FUNCTION_BLOCK FB_Zuiger
VAR_INPUT
	i_eState 			: eSingleState;
	i_eModes			: eModus;
	i_xMoveCiliderDown	: BOOL;
	i_xHallSensorIn		: BOOL;
	i_xHallSensorOut	: BOOL;
	i_xEndSwitchIn		: BOOL;
	i_xEndSwitchOut		: BOOL;
	i_rPressureSensor	: REAL; 
	i_xAlarmResetCilinder	: BOOL;
	i_xAlarmResetAlarmHorizontalMovement	: BOOL;
	i_xAlarmResetPressure : BOOL;
	i_xButtonManStopall : BOOL;
	eManCiliderPosition		: eZuigerCilinderposition;
	eManHorizotalPosition	: eZuigerHorizontaal;
	i_xButtonManVacumOn	: BOOL;
END_VAR
VAR_OUTPUT
	o_xMotor 					: BOOL := FALSE;
	o_xMotorDirectionOut		: BOOL;
	o_xErrorHorizontalMovement 	: BOOL := FALSE;
	o_xAlarmHorizontalMovement	: BOOL;
	o_xMagnetValveCilinder		: BOOL := FALSE;
	o_xMagnetValveVacum	: 			BOOL := FALSE;
	o_xErrorCilinder			: BOOL := FALSE;
	o_xAlarmCilinder			: BOOL;
	o_xErrorPressure			: BOOL := FALSE;
	o_xAlarmPressure			: BOOL;
	o_eCiliderPosition			: eZuigerCilinderposition;
	o_eHorizotalPosition		: eZuigerHorizontaal;
END_VAR
VAR
	eWistedCiliderPosition		: eZuigerCilinderposition;
	eWistedHorizotalPosition	: eZuigerHorizontaal;
	istepcycel : INT;
	TimerCilinder : TON;
	timTimerValue : TIME := T#10S;
	xTimerCilinderRunning: BOOL;
	TimerHorizontal : TON;
	xTimerHorizontalRunning: BOOL;
	
	rPressure_bar: REAL ;
	rMaxbarsensor: REAL := 6;
	rlowpressure: REAL := 4;
	
	
	SIMFUNCTIONING : BOOL := 1;
	o_sStateString: STRING(30);
END_VAR

//Timers
TimerCilinder(IN:=xTimerCilinderRunning, PT := timTimerValue);
TimerHorizontal(IN:=xTimerHorizontalRunning, PT := timTimerValue);
CASE i_eModes OF
	eModus.Off:
		StopALL(); //stopall
	eModus.Auto:
		//Case state + control
		CASE i_eState OF
		eSingleState.Aborting:
			StopALL(); //stopall
		eSingleState.Aborted:
			StopALL(); //stopall
		eSingleState.Execute:
			IF i_xMoveCiliderDown=1 AND istepcycel=0 THEN
				istepcycel:=1;
			END_IF
			IF 	o_xAlarmPressure=0 THEN
				CompleetCycel(); //do a compleet cycel
			END_IF
		eSingleState.Idle:
			istepcycel:=0;
			CiliderUP(); //to startingpostion
			IF o_eCiliderPosition = eZuigerCilinderposition.Up THEN
				HorizontalIN();
			END_IF
		eSingleState.Stopping:
			istepcycel:=0;
			CiliderUP(); //to startingpostion
			IF o_eCiliderPosition = eZuigerCilinderposition.Up THEN
				HorizontalIN();
			END_IF
		eSingleState.Stopped:
			istepcycel:=0;
			CiliderUP(); //to startingpostion
			IF o_eCiliderPosition = eZuigerCilinderposition.Up THEN
				HorizontalIN();
			END_IF
		eSingleState.Suspending:
			istepcycel:=0;
			CiliderUP(); //to startingpostion
			IF o_eCiliderPosition = eZuigerCilinderposition.Up THEN
				HorizontalIN();
			END_IF
		eSingleState.Suspended:
			istepcycel:=0;
			CiliderUP(); //to startingpostion
			IF o_eCiliderPosition = eZuigerCilinderposition.Up THEN
				HorizontalIN();
			END_IF
		END_CASE
	eModus.Manual: //manual controll
		IF i_xButtonManStopall THEN
			StopALL(); //stopall
		ELSIF eManCiliderPosition =  eZuigerCilinderposition.up THEN
			CiliderUP(); //to startingpostion
		ELSIF eManCiliderPosition =  eZuigerCilinderposition.Down THEN
			CilinderDOwn();
		END_IF
		IF NOT i_xButtonManStopall AND eManHorizotalPosition	= eZuigerHorizontaal.In THEN
			HorizontalIN();
		ELSIF NOT i_xButtonManStopall AND eManHorizotalPosition	= eZuigerHorizontaal.Out THEN
			HoriztalOUT();
		END_IF
		IF NOT i_xButtonManStopall AND NOT i_xButtonManVacumOn THEN
			o_xMagnetValveVacum:=FALSE;
		ELSIF NOT i_xButtonManStopall AND i_xButtonManVacumOn THEN
			o_xMagnetValveVacum:=TRUE;
		END_IF
END_CASE

//Errors
IF  NOT (eWistedCiliderPosition = o_eCiliderPosition) THEN //error timer cilinder
	xTimerCilinderRunning:=1;
ELSE
	xTimerCilinderRunning:=0;
END_IF

IF TimerCilinder.Q THEN //error cilinder when timer gone
	o_xErrorCilinder:=1;
	o_xAlarmCilinder:=1;
ELSE
	o_xErrorCilinder:=0;
END_IF

IF  (NOT (eWistedHorizotalPosition = o_eHorizotalPosition)) AND o_xMotor THEN //error start timer horizonal
	xTimerHorizontalRunning:=1;
ELSE
	xTimerHorizontalRunning:=0;
END_IF

IF TimerHorizontal.Q THEN
	o_xErrorHorizontalMovement:=1;
	o_xAlarmHorizontalMovement:=1;
ELSE
	o_xErrorHorizontalMovement:=0;
END_IF

//pressuresensor error
rPressure_bar := (i_rPressureSensor / 4095.0) * rMaxbarsensor;// 4095 form analog and 6 from 6 bar max from the sensor
IF rPressure_bar<rlowpressure THEN
	o_xErrorPressure:=1;
	o_xAlarmPressure:=1;
ELSE
	o_xErrorPressure:=0;
END_IF

//Alarm reset
IF i_xAlarmResetCilinder AND NOT  o_xErrorCilinder THEN
	o_xAlarmCilinder:=0;
END_IF 
IF NOT 	o_xErrorHorizontalMovement AND i_xAlarmResetAlarmHorizontalMovement THEN
	o_xAlarmHorizontalMovement:=0;
END_IF
IF NOT o_xErrorPressure AND  i_xAlarmResetPressure THEN
	o_xAlarmPressure:=0;
END_IF

//actualpostioncilinder
IF	i_xHallSensorIn AND i_xHallSensorOut THEN
	o_eCiliderPosition := eZuigerCilinderposition.Unkown;
ELSIF i_xHallSensorIn	THEN
	o_eCiliderPosition := eZuigerCilinderposition.Up;
ELSIF i_xHallSensorOut THEN
	o_eCiliderPosition := eZuigerCilinderposition.Down;
ELSE
	o_eCiliderPosition := eZuigerCilinderposition.Unkown;
END_IF

//actualpostionhorizontal with motor controll
IF	i_xEndSwitchIn AND i_xEndSwitchOut THEN
	o_eHorizotalPosition := eZuigerHorizontaal.Unkown;
ELSIF i_xEndSwitchIn	THEN
	o_eHorizotalPosition := eZuigerHorizontaal.In;
ELSIF i_xEndSwitchOut THEN
	o_eHorizotalPosition := eZuigerHorizontaal.Out;
ELSE
	o_eHorizotalPosition := eZuigerHorizontaal.Unkown;
END_IF

IF eWistedHorizotalPosition = o_eHorizotalPosition THEN
	o_xMotor:=0;
ELSIF NOT (eWistedHorizotalPosition = o_eHorizotalPosition) THEN
	o_xMotor:=1;
END_IF

SIM();
o_sStateString := F_StateEnumToStringSingleState(i_eState);

METHOD PRIVATE CiliderUP
//moves the cilider up
eWistedCiliderPosition :=eZuigerCilinderposition.Up;
o_xMagnetValveCilinder:=0;
END_METHOD

METHOD PRIVATE CilinderDOwn
VAR_INPUT
END_VAR
//moves the cilider Down
eWistedCiliderPosition :=eZuigerCilinderposition.Down;
o_xMagnetValveCilinder:=1;
END_METHOD

METHOD PRIVATE CompleetCycel
VAR

END_VAR
	o_eHorizotalPosition := eZuigerHorizontaal.In;
		o_eCiliderPosition := eZuigerCilinderposition.Unkown;
		

CASE istepcycel OF
	1: //too startingpostition
		o_xMagnetValveVacum:=FALSE;
		CiliderUP();
		IF o_eCiliderPosition = eZuigerCilinderposition.Up THEN
			HorizontalIN();
		END_IF
		IF o_eCiliderPosition = eZuigerCilinderposition.Up AND o_eHorizotalPosition =eZuigerHorizontaal.IN THEN
			istepcycel:=2;
		END_IF
	2: 		//zuiger naar beneden totdat beneden
		o_xMagnetValveVacum:=TRUE;
		CilinderDOwn();
		IF o_eCiliderPosition = eZuigerCilinderposition.DOWN THEN
			istepcycel:=3;
		END_IF
	3: //zuiger omhoog
		o_xMagnetValveVacum:=TRUE;
		CiliderUP();
		IF o_eCiliderPosition = eZuigerCilinderposition.UP THEN
			istepcycel:=4;
		END_IF
	4:
		o_xMagnetValveVacum:=TRUE;
		HoriztalOUT();
		IF o_eHorizotalPosition = eZuigerHorizontaal.OUT THEN
				istepcycel:=5;
		END_IF
	5:	
		o_xMagnetValveVacum:=FALSE;
		HorizontalIN();
		IF o_eHorizotalPosition = eZuigerHorizontaal.IN THEN
				istepcycel:=0;
		END_IF

END_CASE
END_METHOD

METHOD PRIVATE HorizontalIN
VAR_INPUT
END_VAR

o_xMotorDirectionOut:=0;
eWistedHorizotalPosition := eZuigerHorizontaal.In;
END_METHOD

METHOD PRIVATE HoriztalOUT
VAR_INPUT
END_VAR
//hoizontal out


o_xMotorDirectionOut:=1;
eWistedHorizotalPosition := eZuigerHorizontaal.Out;
END_METHOD

METHOD SIM
VAR

END_VAR
//simulatie
IF gvl.g_xSimulationActive THEN
	IF SIMFUNCTIONING THEN
		

		IF GVL.TimerShort.Q THEN
			i_rPressureSensor := 4000;
			IF o_xMagnetValveCilinder THEN //simulation
				i_xHallSensorIn := FALSE;
				i_xHallSensorOut := TRUE;
			ELSIF NOT o_xMagnetValveCilinder THEN
				i_xHallSensorIn := TRUE;
				i_xHallSensorOut := FALSE;
			END_IF
		END_IF
		
		IF GVL.Timerlong.Q THEN		
			IF o_xMotor AND o_xMotorDirectionOut THEN
				i_xEndSwitchIn := FALSE;
				i_xEndSwitchOut := TRUE;
			ELSIF o_xMotor AND NOT o_xMotorDirectionOut THEN
				i_xEndSwitchIn := TRUE;
				i_xEndSwitchOut := FALSE;
			END_IF
		END_IF
		
	END_IF
	
END_IF
END_METHOD

METHOD PRIVATE StopALL : BOOL
VAR_INPUT
END_VAR
o_xMagnetValveCilinder:=0;
eWistedHorizotalPosition := o_eHorizotalPosition;

IF	i_xHallSensorIn AND i_xHallSensorOut THEN
	o_eCiliderPosition := eZuigerCilinderposition.Unkown;
ELSIF i_xHallSensorIn	THEN
	o_eCiliderPosition := eZuigerCilinderposition.Up;
ELSIF i_xHallSensorOut THEN
	o_eCiliderPosition := eZuigerCilinderposition.Down;
ELSE
	o_eCiliderPosition := eZuigerCilinderposition.Unkown;
END_IF
//i want to dont like this
//eWistedHorizotalPosition = o_eHorizotalPosition;

IF	i_xEndSwitchIn AND i_xEndSwitchOut THEN
	o_eHorizotalPosition := eZuigerHorizontaal.Unkown;
ELSIF i_xEndSwitchIn	THEN
	o_eHorizotalPosition := eZuigerHorizontaal.In;
ELSIF i_xEndSwitchOut THEN
	o_eHorizotalPosition := eZuigerHorizontaal.Out;
ELSE
	o_eHorizotalPosition := eZuigerHorizontaal.Unkown;
END_IF
END_METHOD

END_FUNCTION_BLOCK

(* stored: Version 1.1.0.1
   POU FB_Zuiger: Id {c519e80b-b9ab-471b-ad59-905255fb6490}, SpecialFunc None
   Method CiliderUP: Id {2152594d-2447-4cf4-aa5e-fc79df202b7a}
   Method CilinderDOwn: Id {89ebc8b5-8ad9-4bf6-bf97-7b54cfc097e2}
   Method CompleetCycel: Id {220ffaa2-661c-4b74-ae88-9f0bbe634114}
   Method HorizontalIN: Id {37631e61-4f18-4725-a55a-98346cee9f06}
   Method HoriztalOUT: Id {f2ee4e78-7768-43e6-82bf-d5e0f38931a0}
   Method SIM: Id {bd495253-70b8-4bb0-8434-9bfdfc38d540}
   Method StopALL: Id {a7b526ea-bf90-4b58-9c21-d53d1f796b35} *)
